// TIA Portal V19 export
TYPE "PositioningMachine_CIn"
// stored: Access Published
   STRUCT
      Manager : "PositioningMachine_Manager";
      SOS_Enable : Bool;
      Bwd_ExtEnable : Bool := TRUE;
      Fwd_ExtEnable : Bool := TRUE;
      EnableManChangeVel : Bool := TRUE;   // Enable working of Manual velocity change Low to High
      ExternalAlarms : Bool := FALSE;
      PositionLimits : Struct
         EnableMin : Bool := FALSE;
         PosMin : LReal := 999999999999.0;
         EnableMax : Bool := FALSE;
         PosMax : LReal := -999999999999.0;
      END_STRUCT;
      VelocityOverride : Struct
         Enable : Bool := FALSE;
         Value : LReal := 100.0;   // %
      END_STRUCT;
      TorqueLimits : Struct
         Enable : Bool := FALSE;
         Value : LReal := 100.0;
      END_STRUCT;
      TOParameters : Struct
         DataPresence : Bool;
         Data : "PositioningMachine_Ax_Parameters";
      END_STRUCT;
   END_STRUCT;
END_TYPE
